Yaskawa INFORM job: SERVICE_POS_ST.JBI

/JOB
//NAME SERVICE_POS_ST
//POS
///NPOS 4,0,0,0,0,0
///TOOL 0
///POSTYPE PULSE
///PULSE
C00000=142526,-8517,3700,5815,-74421,-9941
C00001=94187,-12098,-17057,-8831,-64303,14452
C00002=103764,-13557,-29929,10157,-57452,-17266
C00003=79080,26895,-6245,21615,-60536,-42000
//INST
///DATE 2021/10/11 09:29
///ATTR SC,RW
///GROUP1 RB1
NOP
MOVJ C00000 PL=8
MOVJ C00001 PL=8
MOVJ C00002 PL=8
MOVJ C00003 PL=8
END
